TYPE ST_BaseHMIConnectorEvents_ListToDisplay :
STRUCT
END_STRUCT
END_TYPE

(* stored: Version 1.1.0.1
   DUT ST_BaseHMIConnectorEvents_ListToDisplay: Id {a76f8388-425a-0985-338a-d3a600172d4b} *)
